(* PLC project Senza_nome, Sconosciuto Senza_nome 1 *)
(* stored: creationDateTime 2021-04-20T16:49:38, modificationDateTime 2021-04-20T18:22:57 *)

PROGRAM main
  VAR_EXTERNAL
    moneta : BOOL;
    SA : BOOL;
    SB : BOOL;
    aperto : BOOL;
    BLOCCA : BOOL;
    SBLOCCA : BOOL;
  END_VAR
  VAR  (* added by the conversion: wires and edge detectors of the diagram *)
    R_TRIG1 : R_TRIG;
  END_VAR

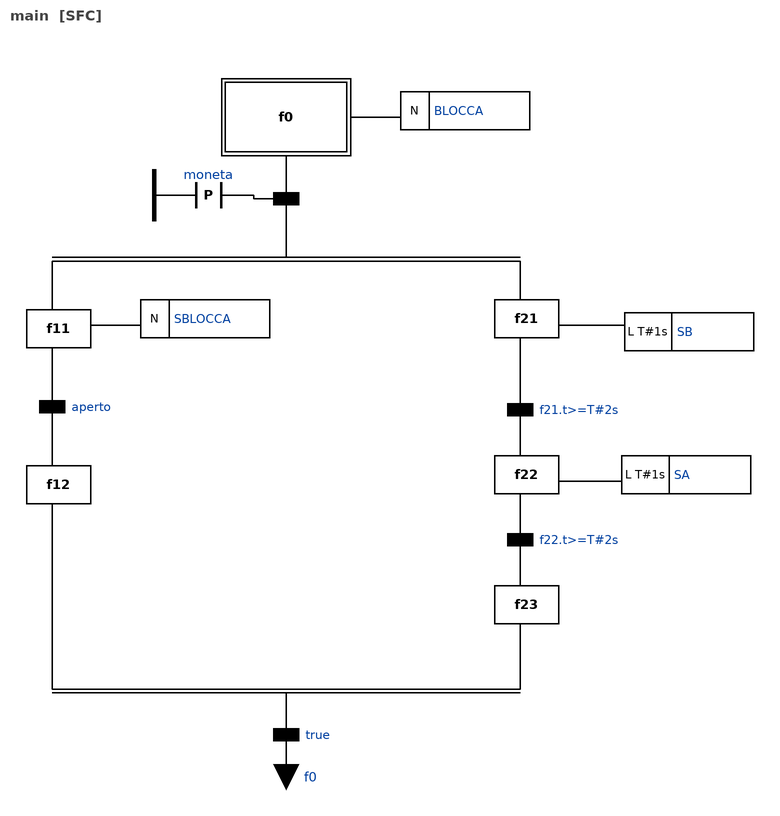
INITIAL_STEP f0:
  BLOCCA(N);
  COMPUTE_FUNCTION_BLOCKS(S);
END_STEP
TRANSITION FROM f0 TO (f11, f21)
  := R_TRIG1.Q;
END_TRANSITION
STEP f21:
  SB(L, T#1s);
END_STEP
TRANSITION FROM f21 TO f22
  := f21.t>=T#2s;
END_TRANSITION
STEP f11:
  SBLOCCA(N);
END_STEP
TRANSITION FROM f11 TO f12
  := aperto;
END_TRANSITION
STEP f22:
  SA(L, T#1s);
END_STEP
TRANSITION FROM f22 TO f23
  := f22.t>=T#2s;
END_TRANSITION
STEP f12:
END_STEP
TRANSITION FROM (f12, f23) TO f0
  := true;
END_TRANSITION
STEP f23:
END_STEP
ACTION COMPUTE_FUNCTION_BLOCKS:  (* blocks drawn on the SFC sheet *)
  R_TRIG1(CLK := moneta);
END_ACTION
END_PROGRAM

FUNCTION_BLOCK distributore
  VAR_INPUT
    attiva_SA : BOOL;  (* Sposta una bibita nel buffer *)
    eroga_prodotto : BOOL;  (* Eroga una bibita *)
    ricarica_prodotto : BOOL;  (* Ricarica 10 bibite nel distributore *)
    preleva : BOOL;  (* Preleva tutte le bibite dal vano prelievo *)
    svuota : BOOL;  (* Sposta tutti i prodotti nel vano di prelievo *)
  END_VAR
  VAR_OUTPUT
    prodotti_da_prelevare : INT := 0;  (* Numero di prodotti nel vano di prelievo *)
    prodotti_disp : BOOL;  (* Prodotto disponibile nel buffer *)
  END_VAR
  VAR
    n_prodotti : INT := 10;  (* Numero di prodotti disponibili *)
    prodotti_buffer : BOOL;  (* Prodotto disponibile nel buffer *)
    eroga_trig : BOOL;  (* Riconoscimento fronte erogazione prodotto *)
    buffer_trig : BOOL;  (* Riconoscimento fronte spostamento prodotto nel buffer *)
    RTRIG_eroga : R_TRIG;
    RTRIG_buffer : R_TRIG;
  END_VAR

            (* Verifica che sia presente almeno un prodotto *)
prodotti_disp := GT(IN1 := n_prodotti,IN2 := 0);

(* Riconoscimento fronte di salita per erogazione prodotto *)
RTRIG_eroga(
     CLK := eroga_prodotto(*BOOL*),
     Q => eroga_trig(*BOOL*));
RTRIG_buffer(
     CLK := attiva_SA(*BOOL*),
     Q => buffer_trig(*BOOL*));
         
(* Sposta prodotto nel buffer se disponibile *)
IF buffer_trig AND prodotti_disp THEN
  n_prodotti := n_prodotti - 1;
  prodotti_buffer := true;
END_IF;

(* Eroga un prodotto se presente nel buffer *)
IF eroga_trig AND prodotti_buffer THEN
  prodotti_buffer := false;
  prodotti_da_prelevare := prodotti_da_prelevare + 1;
END_IF;

(* Ricarica il distributore *)
IF ricarica_prodotto THEN
  n_prodotti := 10;
END_IF;

(* Preleva tutti i prodotti dal vano *)
IF preleva THEN
  prodotti_da_prelevare := 0;
END_IF;

(* Sposta tutti i prodotti nel vano prelievo *)
IF svuota THEN
  prodotti_da_prelevare := prodotti_da_prelevare + n_prodotti;
  n_prodotti := 0;
END_IF;
          
END_FUNCTION_BLOCK

FUNCTION_BLOCK pistone
  VAR_INPUT
    apri : BOOL;  (* Comando di apertura *)
  END_VAR
  VAR_OUTPUT
    aperto : BOOL := 0;  (* Variabile che indica l'avvenuta apertura *)
  END_VAR
  VAR
    TON0 : TON;
    TON1 : TON;
  END_VAR

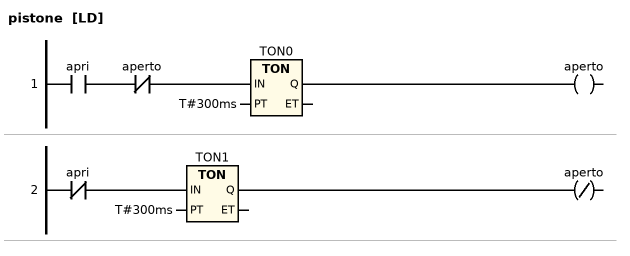
(* LD diagram, written out as Structured Text *)
TON0(IN := apri AND NOT aperto, PT := T#300ms);
aperto := TON0.Q;
TON1(IN := NOT apri, PT := T#300ms);
aperto := NOT TON1.Q;
END_FUNCTION_BLOCK

PROGRAM simulator
  VAR_EXTERNAL
    moneta : BOOL;
    SB : BOOL;
    SA : BOOL;
    SBLOCCA : BOOL;
    BLOCCA : BOOL;
    aperto : BOOL;
  END_VAR
  VAR
    A_aperto : BOOL;  (* Pistone A ritratto *)
    B_aperto : BOOL;  (* Pistone B ritratto *)
    preleva_prodotto : BOOL;  (* Comando preleva prodotto *)
    ricarica_prodotto : BOOL;  (* Comando ricarica distributore *)
    credito_disponibile : BOOL;  (* Comando ricarica distributore *)
    prodotti_nel_vano : INT;  (* Prodotti nel vano di prelievo *)
    prodotti_disponibili : BOOL;  (* Prodotti nel vano di prelievo *)
    distributore0 : distributore;
    pistone0 : pistone;  (* Pistone A *)
    pistone1 : pistone;  (* Pistone B *)
  END_VAR
  VAR  (* added by the conversion: wires and edge detectors of the diagram *)
    R_TRIG1 : R_TRIG;
    R_TRIG2 : R_TRIG;
    R_TRIG3 : R_TRIG;
  END_VAR

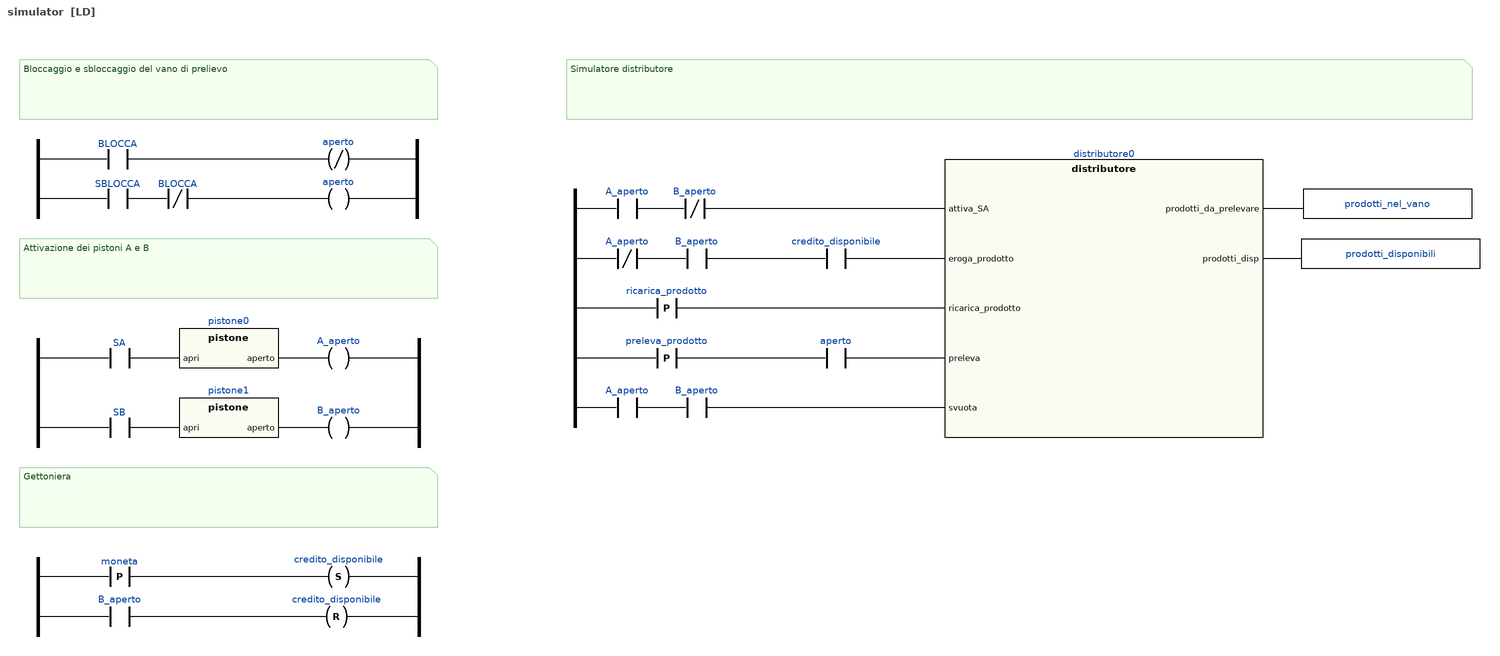
(* LD diagram, written out as Structured Text *)
(* Bloccaggio e sbloccaggio del vano di prelievo *)
(* Simulatore distributore *)
aperto := NOT BLOCCA;
aperto := SBLOCCA AND NOT BLOCCA;
R_TRIG1(CLK := ricarica_prodotto);
R_TRIG2(CLK := preleva_prodotto);
distributore0(attiva_SA := A_aperto AND NOT B_aperto, eroga_prodotto := NOT A_aperto AND B_aperto AND credito_disponibile, ricarica_prodotto := R_TRIG1.Q, preleva := R_TRIG2.Q AND aperto, svuota := A_aperto AND B_aperto);
prodotti_nel_vano := distributore0.prodotti_da_prelevare;
(* Attivazione dei pistoni A e B *)
prodotti_disponibili := distributore0.prodotti_disp;
pistone0(apri := SA);
A_aperto := pistone0.aperto;
pistone1(apri := SB);
B_aperto := pistone1.aperto;
(* Gettoniera *)
R_TRIG3(CLK := moneta);
IF R_TRIG3.Q THEN credito_disponibile := TRUE; END_IF;
IF B_aperto THEN credito_disponibile := FALSE; END_IF;
END_PROGRAM

CONFIGURATION Config0
  RESOURCE Res0 ON PLC
    VAR_GLOBAL
      moneta : BOOL;
      aperto : BOOL;
      SA : BOOL;
      SB : BOOL;
      BLOCCA : BOOL;
      SBLOCCA : BOOL;
    END_VAR
    TASK task0(INTERVAL := T#20ms, PRIORITY := 0);
    PROGRAM instance0 WITH task0 : main;
    PROGRAM instance1 WITH task0 : simulator;
  END_RESOURCE
END_CONFIGURATION
